FUNCTION_BLOCK mqttCommunication IMPLEMENTS ITF_MQTTTool
VAR
	_messageSent : string;
END_VAR

METHOD SendMQTTMessage : BOOL
VAR_INPUT
	Status : STRING;
END_VAR
_messageSent := Status;
END_METHOD

END_FUNCTION_BLOCK

(* stored: Version 1.1.0.1, ProductVersion 3.1.4024.12
   POU mqttCommunication: Id {2ea2534d-2221-4e83-a860-df9cd3f5f013}, SpecialFunc None
   Method SendMQTTMessage: Id {d9bb83be-ccfe-4574-afd2-a18756318aa3} *)
